// TIA Portal V19 export
DATA_BLOCK "instanceR_H_Sys_Status_DB"   // DB28
// stored: InstanceOfName R_H_Sys_Status, InstanceOfType FB
"R_H_Sys_Status"
   // VAR_INPUT
   //    laddrPLC1 : HW_ANY;
   //    laddrPLC2 : HW_ANY;
   //    laddrSystem : HW_ANY;
   //    laddrProfinetPLC1 : HW_ANY;
   //    laddrProfinetPLC2 : HW_ANY;
   // END_VAR
   // VAR_OUTPUT
   //    primaryId : Int;
   //    operationStatePLC1 : UInt;
   //    operationStatePLC2 : UInt;
   //    operationStateSystem : UInt;
   //    mrpRingState : UInt;
   // END_VAR
   // VAR
   //    statDiagModeCpu1 { S7_SetPoint := 'True'} : UInt;
   //    statCountDiagDetailsCpu1 : UInt;
   //    statReturnValueCpu1 : Int;
   //    statDiagCpu1 { ExternalAccessible := 'False'; ExternalVisible := 'False'; ExternalWritable := 'False'; S7_SetPoint := 'True'} : DIS;
   //    statDiagModeCpu2 { S7_SetPoint := 'True'} : UInt;
   //    statCountDiagDetailsCpu2 : UInt;
   //    statReturnValueCpu2 : Int;
   //    statDiagCpu2 { ExternalAccessible := 'False'; ExternalVisible := 'False'; ExternalWritable := 'False'; S7_SetPoint := 'True'} : DIS;
   //    statDiagModeSystem { S7_SetPoint := 'True'} : UInt;
   //    statCountDiagDetailsSystem : UInt;
   //    statReturnValueSystem : Int;
   //    statDiagSystem { ExternalAccessible := 'False'; ExternalVisible := 'False'; ExternalWritable := 'False'; S7_SetPoint := 'True'} : DIS;
   //    statDataRecord1 { S7_SetPoint := 'True'} : "LPNDR_typeMrpInformation";
   //    statDataRecord2 { S7_SetPoint := 'True'} : "LPNDR_typeMrpInformation";
   //    statLPNDR_ReadMrpState { S7_SetPoint := 'True'} : HW_ANY;
   //    statLPNDR_ReadGlobalInfo_DB1 { S7_SetPoint := 'True'} : "LPNDR_ReadGlobalInfo";
   //    statLPNDR_ReadGlobalInfo_DB2 { S7_SetPoint := 'True'} : "LPNDR_ReadGlobalInfo";
   //    statLPNDR_ReadMrpState_DB { S7_SetPoint := 'True'} : "LPNDR_ReadMrpState";
   //    statExecuteClock : Bool;
   //    IEC_Timer_0_Instance { S7_SetPoint := 'True'} : TOF_TIME;
   //    statToggleExecuteClock { S7_SetPoint := 'True'} : Bool;
   //    statUndefinedState : Bool;
   //    statExecuteClock2 : Bool;
   //    statToggleExecuteClock2 : Bool;
   //    IEC_Timer_0_Instance_1 { S7_SetPoint := 'True'} : TOF_TIME;
   //    IEC_Timer_0_Instance_2 { S7_SetPoint := 'True'} : TOF_TIME;
   //    statError1 : Bool;
   //    statChoose1 : Bool;
   //    IEC_Timer_0_Instance_3 { S7_SetPoint := 'True'} : TOF_TIME;
   //    statError2 : Bool;
   //    statChoose2 : Bool;
   // END_VAR
BEGIN
END_DATA_BLOCK
